// ---- VISUs/AxisControl.TcVIS
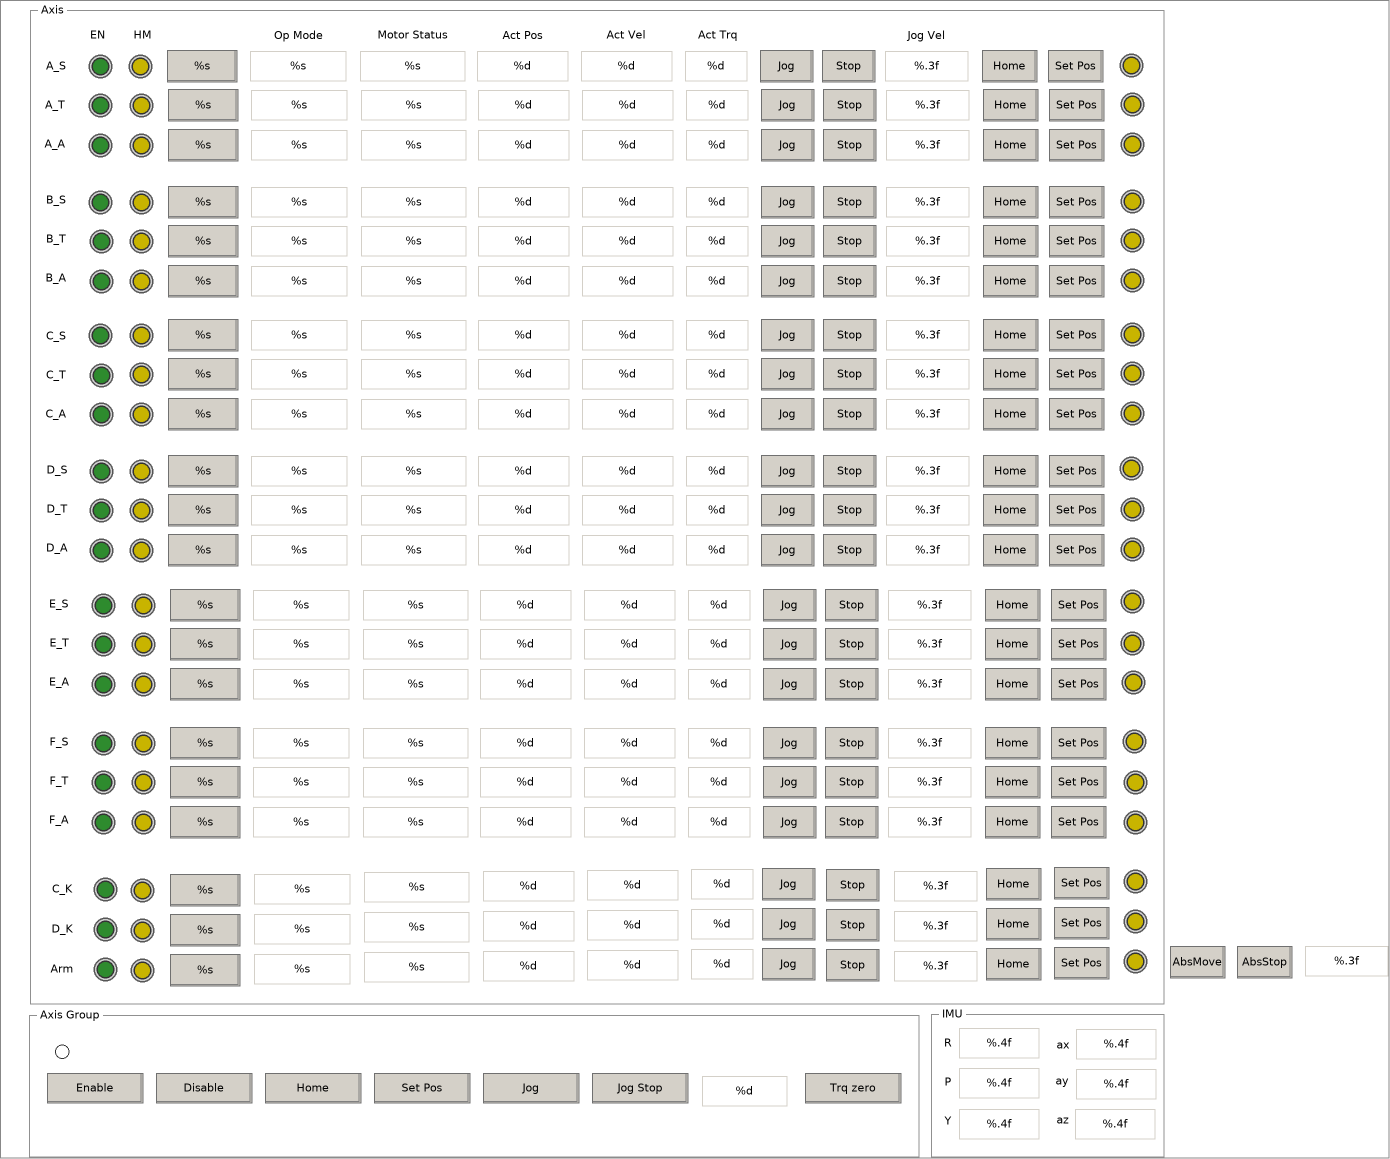
VISUALIZATION AxisControl  // 1390x1159
    GroupBox (30,2 1134x1002), "Axis"
        Label (37,23 61x20), "EN"
        Label (324,25 117x16), "Motor Status"
        Label (239,24 59x19), "Op Mode"
        Label (465,27 55x13), "Act Pos"
        Lamp1 (57,50 27x29), variable: GVL.motorDrive[0].enableBit, style: Lamp-Lamp1-Green
        Textfield (220,49 96x30), "%s", text variable: GVL.motorDrive[0].opModeDispStr
        Textfield (330,49 105x30), "%s", text variable: GVL.motorDrive[0].statusDispStr
        Textfield (447,49 91x30), "%d", text variable: GVL.motorDrive[0].motor.actualPos
        Textfield (551,49 91x30), "%d", text variable: GVL.motorDrive[0].motor.actualVel
        Label (653,25 70x16), "Act Trq"
        Textfield (655,49 62x30), "%d", text variable: GVL.motorDrive[0].motor.actualTrq
        Button (137,48 70x32), "%s", text variable: GVL.enablebuttonText[0]
            toggle GVL.enableButton[0]
        Label (561,25 70x16), "Act Vel"
        Lamp1 (97,50 27x29), variable: GVL.motorDrive[0].isHomeSwitchOn, style: Lamp-Lamp1-Yellow
        Label (91,21 43x24), "HM"
        Button (730,48 53x32), "Jog"
            toggle GVL.jogButton[0]
        Label (869,27 55x13), "Jog Vel"
        Button (952,48 55x32), "Home"
            toggle GVL.startHomeButton[0]
        Button (1018,48 55x32), "Set Pos"
            toggle GVL.setInitPositionButton[0]
        Label (5,54 42x20), "A_S"
        Textfield (855,49 83x30), "%.3f", text variable: GVL.jogVelocity[0]
            OnMouseClick: write the text variable via Default
        Lamp1 (57,89 27x29), variable: GVL.motorDrive[1].enableBit, style: Lamp-Lamp1-Green
        Lamp1 (57,129 27x29), variable: GVL.motorDrive[2].enableBit, style: Lamp-Lamp1-Green
        Lamp1 (57,186 27x29), variable: GVL.motorDrive[3].enableBit, style: Lamp-Lamp1-Green
        Lamp1 (57,319 27x29), variable: GVL.motorDrive[6].enableBit, style: Lamp-Lamp1-Green
        Button (792,48 53x32), "Stop"
            toggle GVL.jogStopButton[0]
        Lamp1 (1088,49 27x29), variable: GVL.motorDrive[0].isHoming, style: Lamp-Lamp1-Yellow
        Lamp1 (1088,452 27x29), variable: GVL.motorDrive[9].isHoming, style: Lamp-Lamp1-Yellow
        Label (8,592 42x20), "E_S"
        Label (8,631 42x20), "E_T"
        Label (8,670 42x20), "E_A"
        Lamp1 (60,589 27x29), variable: GVL.motorDrive[12].enableBit, style: Lamp-Lamp1-Green
        Textfield (223,588 96x30), "%s", text variable: GVL.motorDrive[12].opModeDispStr
        Textfield (333,588 105x30), "%s", text variable: GVL.motorDrive[12].statusDispStr
        Textfield (450,588 91x30), "%d", text variable: GVL.motorDrive[12].motor.actualPos
        Textfield (554,588 91x30), "%d", text variable: GVL.motorDrive[12].motor.actualVel
        Button (140,587 70x32), "%s", text variable: GVL.enablebuttonText[12]
            toggle GVL.enableButton[12]
        Lamp1 (100,589 27x29), variable: GVL.motorDrive[12].isHomeSwitchOn, style: Lamp-Lamp1-Yellow
        Button (733,587 53x32), "Jog"
            toggle GVL.jogButton[12]
        Button (955,587 55x32), "Home"
            toggle GVL.startHomeButton[12]
        Button (1021,587 55x32), "Set Pos"
            toggle GVL.setInitPositionButton[12]
        Textfield (858,588 83x30), "%.3f", text variable: GVL.jogVelocity[12]
            OnMouseClick: write the text variable via Default
        Lamp1 (60,628 27x29), variable: GVL.motorDrive[13].enableBit, style: Lamp-Lamp1-Green
        Lamp1 (60,668 27x29), variable: GVL.motorDrive[14].enableBit, style: Lamp-Lamp1-Green
        Textfield (223,627 96x30), "%s", text variable: GVL.motorDrive[13].opModeDispStr
        Textfield (333,627 105x30), "%s", text variable: GVL.motorDrive[13].statusDispStr
        Textfield (450,627 91x30), "%d", text variable: GVL.motorDrive[13].motor.actualPos
        Textfield (554,627 91x30), "%d", text variable: GVL.motorDrive[13].motor.actualVel
        Textfield (658,627 62x30), "%d", text variable: GVL.motorDrive[13].motor.actualTrq
        Button (140,626 70x32), "%s", text variable: GVL.enablebuttonText[13]
            toggle GVL.enableButton[13]
        Lamp1 (100,628 27x29), variable: GVL.motorDrive[13].isHomeSwitchOn, style: Lamp-Lamp1-Yellow
        Button (733,626 53x32), "Jog"
            toggle GVL.jogButton[13]
        Button (955,626 55x32), "Home"
            toggle GVL.startHomeButton[13]
        Button (1021,626 55x32), "Set Pos"
            toggle GVL.setInitPositionButton[13]
        Textfield (858,627 83x30), "%.3f", text variable: GVL.jogVelocity[13]
            OnMouseClick: write the text variable via Default
        Textfield (223,667 96x30), "%s", text variable: GVL.motorDrive[14].opModeDispStr
        Textfield (333,667 105x30), "%s", text variable: GVL.motorDrive[14].statusDispStr
        Textfield (450,667 91x30), "%d", text variable: GVL.motorDrive[14].motor.actualPos
        Textfield (554,667 91x30), "%d", text variable: GVL.motorDrive[14].motor.actualVel
        Textfield (658,667 62x30), "%d", text variable: GVL.motorDrive[14].motor.actualTrq
        Button (140,666 70x32), "%s", text variable: GVL.enablebuttonText[14]
            toggle GVL.enableButton[14]
        Lamp1 (100,668 27x29), variable: GVL.motorDrive[14].isHomeSwitchOn, style: Lamp-Lamp1-Yellow
        Button (733,666 53x32), "Jog"
            toggle GVL.jogButton[14]
        Button (955,666 55x32), "Home"
            toggle GVL.startHomeButton[14]
        Button (1021,666 55x32), "Set Pos"
            toggle GVL.setInitPositionButton[14]
        Textfield (858,667 83x30), "%.3f", text variable: GVL.jogVelocity[14]
            OnMouseClick: write the text variable via Default
        Button (795,587 53x32), "Stop"
            toggle GVL.jogStopButton[12]
        Button (795,626 53x32), "Stop"
            toggle GVL.jogStopButton[13]
        Button (795,666 53x32), "Stop"
            toggle GVL.jogStopButton[14]
        Label (8,730 42x20), "F_S"
        Label (8,769 42x20), "F_T"
        Label (8,808 42x20), "F_A"
        Lamp1 (60,727 27x29), variable: GVL.motorDrive[15].enableBit, style: Lamp-Lamp1-Green
        Textfield (223,726 96x30), "%s", text variable: GVL.motorDrive[15].opModeDispStr
        Textfield (333,726 105x30), "%s", text variable: GVL.motorDrive[15].statusDispStr
        Textfield (450,726 91x30), "%d", text variable: GVL.motorDrive[15].motor.actualPos
        Textfield (554,726 91x30), "%d", text variable: GVL.motorDrive[15].motor.actualVel
        Textfield (658,726 62x30), "%d", text variable: GVL.motorDrive[15].motor.actualTrq
        Button (140,725 70x32), "%s", text variable: GVL.enablebuttonText[15]
            toggle GVL.enableButton[15]
        Lamp1 (100,727 27x29), variable: GVL.motorDrive[15].isHomeSwitchOn, style: Lamp-Lamp1-Yellow
        Button (733,725 53x32), "Jog"
            toggle GVL.jogButton[15]
        Button (955,725 55x32), "Home"
            toggle GVL.startHomeButton[15]
        Button (1021,725 55x32), "Set Pos"
            toggle GVL.setInitPositionButton[15]
        Textfield (858,726 83x30), "%.3f", text variable: GVL.jogVelocity[15]
            OnMouseClick: write the text variable via Default
        Lamp1 (60,766 27x29), variable: GVL.motorDrive[16].enableBit, style: Lamp-Lamp1-Green
        Lamp1 (60,806 27x29), variable: GVL.motorDrive[17].enableBit, style: Lamp-Lamp1-Green
        Textfield (223,765 96x30), "%s", text variable: GVL.motorDrive[16].opModeDispStr
        Textfield (333,765 105x30), "%s", text variable: GVL.motorDrive[16].statusDispStr
        Textfield (450,765 91x30), "%d", text variable: GVL.motorDrive[16].motor.actualPos
        Textfield (554,765 91x30), "%d", text variable: GVL.motorDrive[16].motor.actualVel
        Textfield (658,765 62x30), "%d", text variable: GVL.motorDrive[16].motor.actualTrq
        Button (140,764 70x32), "%s", text variable: GVL.enablebuttonText[16]
            toggle GVL.enableButton[16]
        Lamp1 (100,766 27x29), variable: GVL.motorDrive[16].isHomeSwitchOn, style: Lamp-Lamp1-Yellow
        Button (733,764 53x32), "Jog"
            toggle GVL.jogButton[16]
        Button (955,764 55x32), "Home"
            toggle GVL.startHomeButton[16]
        Button (1021,764 55x32), "Set Pos"
            toggle GVL.setInitPositionButton[16]
        Textfield (858,765 83x30), "%.3f", text variable: GVL.jogVelocity[16]
            OnMouseClick: write the text variable via Default
        Textfield (223,805 96x30), "%s", text variable: GVL.motorDrive[17].opModeDispStr
        Textfield (333,805 105x30), "%s", text variable: GVL.motorDrive[17].statusDispStr
        Textfield (450,805 91x30), "%d", text variable: GVL.motorDrive[17].motor.actualPos
        Textfield (554,805 91x30), "%d", text variable: GVL.motorDrive[17].motor.actualVel
        Textfield (658,805 62x30), "%d", text variable: GVL.motorDrive[17].motor.actualTrq
        Button (140,804 70x32), "%s", text variable: GVL.enablebuttonText[17]
            toggle GVL.enableButton[17]
        Lamp1 (100,806 27x29), variable: GVL.motorDrive[17].isHomeSwitchOn, style: Lamp-Lamp1-Yellow
        Button (733,804 53x32), "Jog"
            toggle GVL.jogButton[17]
        Button (955,804 55x32), "Home"
            toggle GVL.startHomeButton[17]
        Button (1021,804 55x32), "Set Pos"
            toggle GVL.setInitPositionButton[17]
        Textfield (858,805 83x30), "%.3f", text variable: GVL.jogVelocity[17]
            OnMouseClick: write the text variable via Default
        Button (795,725 53x32), "Stop"
            toggle GVL.jogStopButton[15]
        Button (795,764 53x32), "Stop"
            toggle GVL.jogStopButton[16]
        Button (795,804 53x32), "Stop"
            toggle GVL.jogStopButton[17]
        Lamp1 (1089,585 27x29), variable: GVL.motorDrive[12].isHoming, style: Lamp-Lamp1-Yellow
        Lamp1 (1091,725 27x29), variable: GVL.motorDrive[15].isHoming, style: Lamp-Lamp1-Yellow
        Lamp1 (1092,766 27x29), variable: GVL.motorDrive[16].isHoming, style: Lamp-Lamp1-Yellow
        Lamp1 (1092,806 27x29), variable: GVL.motorDrive[17].isHoming, style: Lamp-Lamp1-Yellow
        Lamp1 (1089,627 27x29), variable: GVL.motorDrive[13].isHoming, style: Lamp-Lamp1-Yellow
        Label (11,877 42x20), "C_K"
        Lamp1 (62,873 27x29), variable: GVL.motorDrive[18].enableBit, style: Lamp-Lamp1-Green
        Lamp1 (99,874 27x29), variable: GVL.motorDrive[18].isHomeSwitchOn, style: Lamp-Lamp1-Yellow
        Button (140,872 70x32), "%s", text variable: GVL.enablebuttonText[17]
            toggle GVL.enableButton[18]
        Textfield (224,872 96x30), "%s", text variable: GVL.motorDrive[18].opModeDispStr
        Textfield (334,870 105x30), "%s", text variable: GVL.motorDrive[18].statusDispStr
        Textfield (453,869 91x30), "%d", text variable: GVL.motorDrive[18].motor.actualPos
        Textfield (557,868 91x30), "%d", text variable: GVL.motorDrive[18].motor.actualVel
        Textfield (661,867 62x30), "%d", text variable: GVL.motorDrive[18].motor.actualTrq
        Button (732,866 53x32), "Jog"
            toggle GVL.jogButton[18]
        Button (796,867 53x32), "Stop"
            toggle GVL.jogStopButton[18]
        Textfield (864,869 83x30), "%.3f", text variable: GVL.jogVelocity[18]
            OnMouseClick: write the text variable via Default
        Button (956,866 55x32), "Home"
            toggle GVL.startHomeButton[18]
        Button (1024,865 55x32), "Set Pos"
            toggle GVL.setInitPositionButton[18]
        Lamp1 (1092,865 27x29), variable: GVL.motorDrive[18].isHoming, style: Lamp-Lamp1-Yellow
        Textfield (658,588 62x30), "%d", text variable: GVL.motorDrive[12].motor.actualTrq
        Label (11,917 42x20), "D_K"
        Label (11,957 42x20), "Arm"
    Label (34,95 42x20), "A_T"
    Label (34,134 42x20), "A_A"
    Label (35,190 42x20), "B_S"
    Label (35,229 42x20), "B_T"
    Label (35,268 42x20), "B_A"
    Label (35,326 42x20), "C_S"
    Label (35,365 42x20), "C_T"
    Label (35,404 42x20), "C_A"
    Label (36,460 42x20), "D_S"
    Label (36,499 42x20), "D_T"
    Label (36,538 42x20), "D_A"
    GroupBox (29,1007 890x150), "Axis Group"
        RadioButton (24,30 783x29), variable: GVL.groupSelector
            Areas[1]: Text=Shank
            Areas[2]: Text=Thigh
            Areas[3]: Text=Side
            Areas[4]: Text=LegA
            Areas[5]: Text=LegB
            Areas[6]: Text=LegC
            Areas[7]: Text=LegD
            Areas[8]: Text=LegE
            Areas[9]: Text=LegF
        Button (18,66 96x30), "Enable"
            toggle GVL.enableGroupButton
        Button (127,66 96x30), "Disable"
            toggle GVL.disableGroupButton
        Button (236,66 96x30), "Home"
            toggle GVL.homeGroupButton
        Button (345,66 96x30), "Set Pos"
            toggle GVL.setPosGroupButton
        Button (454,66 96x30), "Jog"
            toggle GVL.jogGroupButton
        Button (776,66 96x30), "Trq zero"
            toggle GVL.setTSRZeroButton
        Textfield (673,69 85x30), "%d", text variable: GVL.jogGroupVelocity
            OnMouseClick: write the text variable via Default
        Button (563,66 96x30), "Jog Stop"
            toggle GVL.jogStopGroupButton
    Textfield (251,90 96x30), "%s", text variable: GVL.motorDrive[1].opModeDispStr
    Textfield (361,90 105x30), "%s", text variable: GVL.motorDrive[1].statusDispStr
    Textfield (478,90 91x30), "%d", text variable: GVL.motorDrive[1].motor.actualPos
    Textfield (582,90 91x30), "%d", text variable: GVL.motorDrive[1].motor.actualVel
    Textfield (686,90 62x30), "%d", text variable: GVL.motorDrive[1].motor.actualTrq
    Button (168,89 70x32), "%s", text variable: GVL.enablebuttonText[1]
        toggle GVL.enableButton[1]
    Lamp1 (128,91 27x29), variable: GVL.motorDrive[1].isHomeSwitchOn, style: Lamp-Lamp1-Yellow
    Button (761,89 53x32), "Jog"
        toggle GVL.jogButton[1]
    Button (983,89 55x32), "Home"
        toggle GVL.startHomeButton[1]
    Button (1049,89 55x32), "Set Pos"
        toggle GVL.setInitPositionButton[1]
    Textfield (886,90 83x30), "%.3f", text variable: GVL.jogVelocity[1]
        OnMouseClick: write the text variable via Default
    Textfield (251,130 96x30), "%s", text variable: GVL.motorDrive[2].opModeDispStr
    Textfield (361,130 105x30), "%s", text variable: GVL.motorDrive[2].statusDispStr
    Textfield (478,130 91x30), "%d", text variable: GVL.motorDrive[2].motor.actualPos
    Textfield (582,130 91x30), "%d", text variable: GVL.motorDrive[2].motor.actualVel
    Textfield (686,130 62x30), "%d", text variable: GVL.motorDrive[2].motor.actualTrq
    Button (168,129 70x32), "%s", text variable: GVL.enablebuttonText[2]
        toggle GVL.enableButton[2]
    Lamp1 (128,131 27x29), variable: GVL.motorDrive[2].isHomeSwitchOn, style: Lamp-Lamp1-Yellow
    Button (761,129 53x32), "Jog"
        toggle GVL.jogButton[2]
    Button (983,129 55x32), "Home"
        toggle GVL.startHomeButton[2]
    Button (1049,129 55x32), "Set Pos"
        toggle GVL.setInitPositionButton[2]
    Textfield (886,130 83x30), "%.3f", text variable: GVL.jogVelocity[2]
        OnMouseClick: write the text variable via Default
    Textfield (251,187 96x30), "%s", text variable: GVL.motorDrive[3].opModeDispStr
    Textfield (361,187 105x30), "%s", text variable: GVL.motorDrive[3].statusDispStr
    Textfield (478,187 91x30), "%d", text variable: GVL.motorDrive[3].motor.actualPos
    Textfield (582,187 91x30), "%d", text variable: GVL.motorDrive[3].motor.actualVel
    Textfield (686,187 62x30), "%d", text variable: GVL.motorDrive[3].motor.actualTrq
    Button (168,186 70x32), "%s", text variable: GVL.enablebuttonText[3]
        toggle GVL.enableButton[3]
    Lamp1 (128,188 27x29), variable: GVL.motorDrive[3].isHomeSwitchOn, style: Lamp-Lamp1-Yellow
    Button (761,186 53x32), "Jog"
        toggle GVL.jogButton[3]
    Button (983,186 55x32), "Home"
        toggle GVL.startHomeButton[3]
    Button (1049,186 55x32), "Set Pos"
        toggle GVL.setInitPositionButton[3]
    Textfield (886,187 83x30), "%.3f", text variable: GVL.jogVelocity[3]
        OnMouseClick: write the text variable via Default
    Lamp1 (88,227 27x29), variable: GVL.motorDrive[4].enableBit, style: Lamp-Lamp1-Green
    Lamp1 (88,267 27x29), variable: GVL.motorDrive[5].enableBit, style: Lamp-Lamp1-Green
    Textfield (251,226 96x30), "%s", text variable: GVL.motorDrive[4].opModeDispStr
    Textfield (361,226 105x30), "%s", text variable: GVL.motorDrive[4].statusDispStr
    Textfield (478,226 91x30), "%d", text variable: GVL.motorDrive[4].motor.actualPos
    Textfield (582,226 91x30), "%d", text variable: GVL.motorDrive[4].motor.actualVel
    Textfield (686,226 62x30), "%d", text variable: GVL.motorDrive[4].motor.actualTrq
    Button (168,225 70x32), "%s", text variable: GVL.enablebuttonText[4]
        toggle GVL.enableButton[4]
    Lamp1 (128,227 27x29), variable: GVL.motorDrive[4].isHomeSwitchOn, style: Lamp-Lamp1-Yellow
    Button (761,225 53x32), "Jog"
        toggle GVL.jogButton[4]
    Button (983,225 55x32), "Home"
        toggle GVL.startHomeButton[4]
    Button (1049,225 55x32), "Set Pos"
        toggle GVL.setInitPositionButton[4]
    Textfield (886,226 83x30), "%.3f", text variable: GVL.jogVelocity[4]
        OnMouseClick: write the text variable via Default
    Textfield (251,266 96x30), "%s", text variable: GVL.motorDrive[5].opModeDispStr
    Textfield (361,266 105x30), "%s", text variable: GVL.motorDrive[5].statusDispStr
    Textfield (478,266 91x30), "%d", text variable: GVL.motorDrive[5].motor.actualPos
    Textfield (582,266 91x30), "%d", text variable: GVL.motorDrive[5].motor.actualVel
    Textfield (686,266 62x30), "%d", text variable: GVL.motorDrive[5].motor.actualTrq
    Button (168,265 70x32), "%s", text variable: GVL.enablebuttonText[5]
        toggle GVL.enableButton[5]
    Lamp1 (128,267 27x29), variable: GVL.motorDrive[5].isHomeSwitchOn, style: Lamp-Lamp1-Yellow
    Button (761,265 53x32), "Jog"
        toggle GVL.jogButton[5]
    Button (983,265 55x32), "Home"
        toggle GVL.startHomeButton[5]
    Button (1049,265 55x32), "Set Pos"
        toggle GVL.setInitPositionButton[5]
    Textfield (886,266 83x30), "%.3f", text variable: GVL.jogVelocity[5]
        OnMouseClick: write the text variable via Default
    Textfield (251,320 96x30), "%s", text variable: GVL.motorDrive[6].opModeDispStr
    Textfield (361,320 105x30), "%s", text variable: GVL.motorDrive[6].statusDispStr
    Textfield (478,320 91x30), "%d", text variable: GVL.motorDrive[6].motor.actualPos
    Textfield (582,320 91x30), "%d", text variable: GVL.motorDrive[6].motor.actualVel
    Textfield (686,320 62x30), "%d", text variable: GVL.motorDrive[6].motor.actualTrq
    Button (168,319 70x32), "%s", text variable: GVL.enablebuttonText[6]
        toggle GVL.enableButton[6]
    Lamp1 (128,321 27x29), variable: GVL.motorDrive[6].isHomeSwitchOn, style: Lamp-Lamp1-Yellow
    Button (761,319 53x32), "Jog"
        toggle GVL.jogButton[6]
    Button (983,319 55x32), "Home"
        toggle GVL.startHomeButton[6]
    Button (1049,319 55x32), "Set Pos"
        toggle GVL.setInitPositionButton[6]
    Textfield (886,320 83x30), "%.3f", text variable: GVL.jogVelocity[6]
        OnMouseClick: write the text variable via Default
    Lamp1 (88,361 27x29), variable: GVL.motorDrive[7].enableBit, style: Lamp-Lamp1-Green
    Lamp1 (88,400 27x29), variable: GVL.motorDrive[8].enableBit, style: Lamp-Lamp1-Green
    Lamp1 (88,457 27x29), variable: GVL.motorDrive[9].enableBit, style: Lamp-Lamp1-Green
    Textfield (251,359 96x30), "%s", text variable: GVL.motorDrive[7].opModeDispStr
    Textfield (361,359 105x30), "%s", text variable: GVL.motorDrive[7].statusDispStr
    Textfield (478,359 91x30), "%d", text variable: GVL.motorDrive[7].motor.actualPos
    Textfield (582,359 91x30), "%d", text variable: GVL.motorDrive[7].motor.actualVel
    Textfield (686,359 62x30), "%d", text variable: GVL.motorDrive[7].motor.actualTrq
    Button (168,358 70x32), "%s", text variable: GVL.enablebuttonText[7]
        toggle GVL.enableButton[7]
    Lamp1 (128,360 27x29), variable: GVL.motorDrive[7].isHomeSwitchOn, style: Lamp-Lamp1-Yellow
    Button (761,358 53x32), "Jog"
        toggle GVL.jogButton[7]
    Button (983,358 55x32), "Home"
        toggle GVL.startHomeButton[7]
    Button (1049,358 55x32), "Set Pos"
        toggle GVL.setInitPositionButton[7]
    Textfield (886,359 83x30), "%.3f", text variable: GVL.jogVelocity[7]
        OnMouseClick: write the text variable via Default
    Textfield (251,399 96x30), "%s", text variable: GVL.motorDrive[8].opModeDispStr
    Textfield (361,399 105x30), "%s", text variable: GVL.motorDrive[8].statusDispStr
    Textfield (478,399 91x30), "%d", text variable: GVL.motorDrive[8].motor.actualPos
    Textfield (582,399 91x30), "%d", text variable: GVL.motorDrive[8].motor.actualVel
    Textfield (686,399 62x30), "%d", text variable: GVL.motorDrive[8].motor.actualTrq
    Button (168,398 70x32), "%s", text variable: GVL.enablebuttonText[8]
        toggle GVL.enableButton[8]
    Lamp1 (128,400 27x29), variable: GVL.motorDrive[8].isHomeSwitchOn, style: Lamp-Lamp1-Yellow
    Button (761,398 53x32), "Jog"
        toggle GVL.jogButton[8]
    Button (983,398 55x32), "Home"
        toggle GVL.startHomeButton[8]
    Button (1049,398 55x32), "Set Pos"
        toggle GVL.setInitPositionButton[8]
    Textfield (886,399 83x30), "%.3f", text variable: GVL.jogVelocity[8]
        OnMouseClick: write the text variable via Default
    Textfield (251,456 96x30), "%s", text variable: GVL.motorDrive[9].opModeDispStr
    Textfield (361,456 105x30), "%s", text variable: GVL.motorDrive[9].statusDispStr
    Textfield (478,456 91x30), "%d", text variable: GVL.motorDrive[9].motor.actualPos
    Textfield (582,456 91x30), "%d", text variable: GVL.motorDrive[9].motor.actualVel
    Textfield (686,456 62x30), "%d", text variable: GVL.motorDrive[9].motor.actualTrq
    Button (168,455 70x32), "%s", text variable: GVL.enablebuttonText[9]
        toggle GVL.enableButton[9]
    Lamp1 (128,457 27x29), variable: GVL.motorDrive[9].isHomeSwitchOn, style: Lamp-Lamp1-Yellow
    Button (761,455 53x32), "Jog"
        toggle GVL.jogButton[9]
    Button (983,455 55x32), "Home"
        toggle GVL.startHomeButton[9]
    Button (1049,455 55x32), "Set Pos"
        toggle GVL.setInitPositionButton[9]
    Textfield (886,456 83x30), "%.3f", text variable: GVL.jogVelocity[9]
        OnMouseClick: write the text variable via Default
    Lamp1 (88,496 27x29), variable: GVL.motorDrive[10].enableBit, style: Lamp-Lamp1-Green
    Lamp1 (88,536 27x29), variable: GVL.motorDrive[11].enableBit, style: Lamp-Lamp1-Green
    Textfield (251,495 96x30), "%s", text variable: GVL.motorDrive[10].opModeDispStr
    Textfield (361,495 105x30), "%s", text variable: GVL.motorDrive[10].statusDispStr
    Textfield (478,495 91x30), "%d", text variable: GVL.motorDrive[10].motor.actualPos
    Textfield (582,495 91x30), "%d", text variable: GVL.motorDrive[10].motor.actualVel
    Textfield (686,495 62x30), "%d", text variable: GVL.motorDrive[10].motor.actualTrq
    Button (168,494 70x32), "%s", text variable: GVL.enablebuttonText[10]
        toggle GVL.enableButton[10]
    Lamp1 (128,496 27x29), variable: GVL.motorDrive[10].isHomeSwitchOn, style: Lamp-Lamp1-Yellow
    Button (761,494 53x32), "Jog"
        toggle GVL.jogButton[10]
    Button (983,494 55x32), "Home"
        toggle GVL.startHomeButton[10]
    Button (1049,494 55x32), "Set Pos"
        toggle GVL.setInitPositionButton[10]
    Textfield (886,495 83x30), "%.3f", text variable: GVL.jogVelocity[10]
        OnMouseClick: write the text variable via Default
    Textfield (251,535 96x30), "%s", text variable: GVL.motorDrive[11].opModeDispStr
    Textfield (361,535 105x30), "%s", text variable: GVL.motorDrive[11].statusDispStr
    Textfield (478,535 91x30), "%d", text variable: GVL.motorDrive[11].motor.actualPos
    Textfield (582,535 91x30), "%d", text variable: GVL.motorDrive[11].motor.actualVel
    Textfield (686,535 62x30), "%d", text variable: GVL.motorDrive[11].motor.actualTrq
    Button (168,534 70x32), "%s", text variable: GVL.enablebuttonText[11]
        toggle GVL.enableButton[11]
    Lamp1 (128,536 27x29), variable: GVL.motorDrive[11].isHomeSwitchOn, style: Lamp-Lamp1-Yellow
    Button (761,534 53x32), "Jog"
        toggle GVL.jogButton[11]
    Button (983,534 55x32), "Home"
        toggle GVL.startHomeButton[11]
    Button (1049,534 55x32), "Set Pos"
        toggle GVL.setInitPositionButton[11]
    Textfield (886,535 83x30), "%.3f", text variable: GVL.jogVelocity[11]
        OnMouseClick: write the text variable via Default
    Button (823,89 53x32), "Stop"
        toggle GVL.jogStopButton[1]
    Button (823,129 53x32), "Stop"
        toggle GVL.jogStopButton[2]
    Button (823,186 53x32), "Stop"
        toggle GVL.jogStopButton[3]
    Button (823,225 53x32), "Stop"
        toggle GVL.jogStopButton[4]
    Button (823,265 53x32), "Stop"
        toggle GVL.jogStopButton[5]
    Button (823,319 53x32), "Stop"
        toggle GVL.jogStopButton[6]
    Button (823,358 53x32), "Stop"
        toggle GVL.jogStopButton[7]
    Button (823,398 53x32), "Stop"
        toggle GVL.jogStopButton[8]
    Button (823,455 53x32), "Stop"
        toggle GVL.jogStopButton[9]
    Button (823,494 53x32), "Stop"
        toggle GVL.jogStopButton[10]
    Button (823,534 53x32), "Stop"
        toggle GVL.jogStopButton[11]
    Lamp1 (1119,90 27x29), variable: GVL.motorDrive[1].isHoming, style: Lamp-Lamp1-Yellow
    Lamp1 (1119,130 27x29), variable: GVL.motorDrive[2].isHoming, style: Lamp-Lamp1-Yellow
    Lamp1 (1119,187 27x29), variable: GVL.motorDrive[3].isHoming, style: Lamp-Lamp1-Yellow
    Lamp1 (1119,226 27x29), variable: GVL.motorDrive[4].isHoming, style: Lamp-Lamp1-Yellow
    Lamp1 (1119,266 27x29), variable: GVL.motorDrive[5].isHoming, style: Lamp-Lamp1-Yellow
    Lamp1 (1119,320 27x29), variable: GVL.motorDrive[6].isHoming, style: Lamp-Lamp1-Yellow
    Lamp1 (1119,359 27x29), variable: GVL.motorDrive[7].isHoming, style: Lamp-Lamp1-Yellow
    Lamp1 (1119,399 27x29), variable: GVL.motorDrive[8].isHoming, style: Lamp-Lamp1-Yellow
    Lamp1 (1119,495 27x29), variable: GVL.motorDrive[10].isHoming, style: Lamp-Lamp1-Yellow
    Lamp1 (1119,535 27x29), variable: GVL.motorDrive[11].isHoming, style: Lamp-Lamp1-Yellow
    Lamp1 (1120,668 27x29), variable: GVL.motorDrive[14].isHoming, style: Lamp-Lamp1-Yellow
    GroupBox (931,1006 233x151), "IMU"
        Textfield (28,22 80x30), "%.4f", text variable: GVL.rpy_model[0]
        Textfield (28,62 80x30), "%.4f", text variable: GVL.rpy_model[1]
        Textfield (28,103 80x30), "%.4f", text variable: GVL.rpy_model[2]
        Label (-5,22 44x30), "R"
        Label (-5,61 44x30), "P"
        Label (-5,100 44x30), "Y"
        Textfield (145,23 80x30), "%.4f", text variable: GVL.accx
        Label (110,24 44x30), "ax"
        Textfield (145,63 80x30), "%.4f", text variable: GVL.accy
        Label (109,60 44x30), "ay"
        Label (110,99 44x30), "az"
        Textfield (144,103 80x30), "%.4f", text variable: GVL.accz
    Lamp1 (92,915 27x29), variable: GVL.motorDrive[19].enableBit, style: Lamp-Lamp1-Green
    Lamp1 (129,916 27x29), variable: GVL.motorDrive[19].isHomeSwitchOn, style: Lamp-Lamp1-Yellow
    Button (170,914 70x32), "%s", text variable: GVL.enablebuttonText[17]
        toggle GVL.enableButton[19]
    Textfield (254,914 96x30), "%s", text variable: GVL.motorDrive[19].opModeDispStr
    Textfield (364,912 105x30), "%s", text variable: GVL.motorDrive[19].statusDispStr
    Textfield (483,911 91x30), "%d", text variable: GVL.motorDrive[19].motor.actualPos
    Textfield (587,910 91x30), "%d", text variable: GVL.motorDrive[19].motor.actualVel
    Textfield (691,909 62x30), "%d", text variable: GVL.motorDrive[19].motor.actualTrq
    Button (762,908 53x32), "Jog"
        toggle GVL.jogButton[19]
    Button (826,909 53x32), "Stop"
        toggle GVL.jogStopButton[19]
    Textfield (894,911 83x30), "%.3f", text variable: GVL.jogVelocity[19]
        OnMouseClick: write the text variable via Default
    Button (986,908 55x32), "Home"
        toggle GVL.startHomeButton[19]
    Button (1054,907 55x32), "Set Pos"
        toggle GVL.setInitPositionButton[19]
    Lamp1 (1122,907 27x29), variable: GVL.motorDrive[19].isHoming, style: Lamp-Lamp1-Yellow
    Lamp1 (92,955 27x29), variable: GVL.motorDrive[20].enableBit, style: Lamp-Lamp1-Green
    Lamp1 (129,956 27x29), variable: GVL.motorDrive[20].isHomeSwitchOn, style: Lamp-Lamp1-Yellow
    Button (170,954 70x32), "%s", text variable: GVL.enablebuttonText[17]
        toggle GVL.enableButton[20]
    Textfield (254,954 96x30), "%s", text variable: GVL.motorDrive[20].opModeDispStr
    Textfield (364,952 105x30), "%s", text variable: GVL.motorDrive[20].statusDispStr
    Textfield (483,951 91x30), "%d", text variable: GVL.motorDrive[20].motor.actualPos
    Textfield (587,950 91x30), "%d", text variable: GVL.motorDrive[20].motor.actualVel
    Textfield (691,949 62x30), "%d", text variable: GVL.motorDrive[20].motor.actualTrq
    Button (762,948 53x32), "Jog"
        toggle GVL.jogButton[20]
    Button (826,949 53x32), "Stop"
        toggle GVL.jogStopButton[20]
    Textfield (894,951 83x30), "%.3f", text variable: GVL.jogVelocity[20]
        OnMouseClick: write the text variable via Default
    Button (986,948 55x32), "Home"
        toggle GVL.startHomeButton[20]
    Button (1054,947 55x32), "Set Pos"
        toggle GVL.setInitPositionButton[20]
    Lamp1 (1122,947 27x29), variable: GVL.motorDrive[20].isHoming, style: Lamp-Lamp1-Yellow
    Button (1170,946 55x32), "AbsMove"
        toggle GVL.AbsMoveButton[20]
    Textfield (1305,946 83x30), "%.3f", text variable: GVL.AbsMoveTgtPos[20]
        OnMouseClick: write the text variable via Default
    Button (1237,946 55x32), "AbsStop"
        toggle GVL.AbsMoveStopButton[20]
END_VISUALIZATION

// ---- VISUs/ForceControl.TcVIS
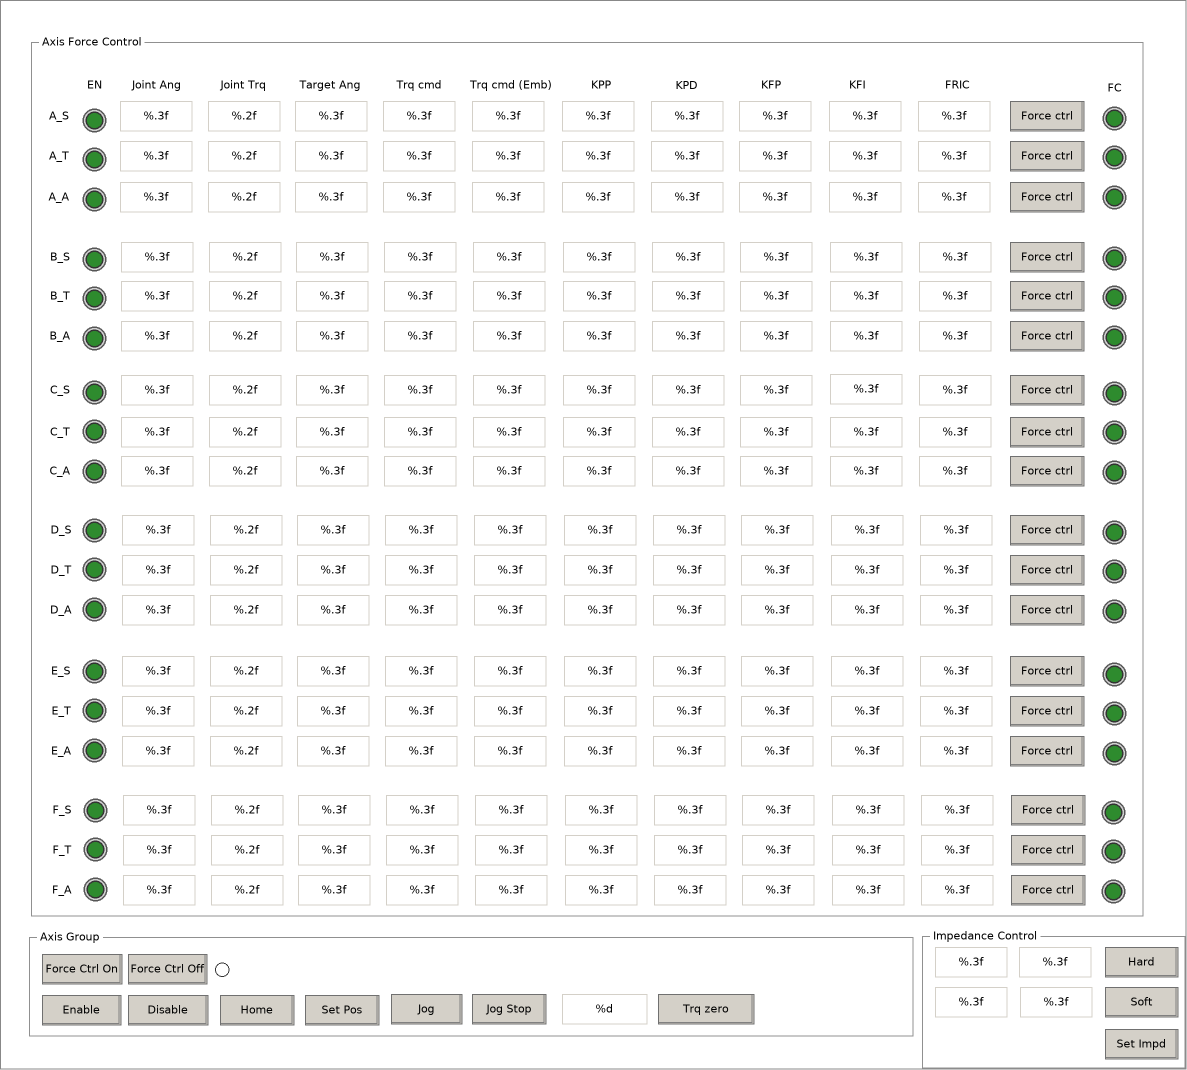
VISUALIZATION ForceControl  // 1187x1070
    GroupBox (31,34 1112x882), "Axis Force Control"
        Label (90,36 71x30), "Joint Ang"
        Label (179,36 67x30), "Joint Trq"
        Label (263,36 72x30), "Target Ang"
        Label (353,36 70x30), "Trq cmd"
        Label (433,36 94x30), "Trq cmd (Emb)"
        Textfield (89,67 72x30), "%.3f", text variable: GVL.motorDrive[0].motorAngle
        Label (545,39 50x24), "KPP"
        Label (632,36 47x31), "KPD"
        Label (800,36 53x30), "KFI"
        Label (714,36 52x30), "KFP"
        Label (900,36 53x30), "FRIC"
        Label (7,72 42x20), "A_S"
        Label (7,112 42x20), "A_T"
        Label (7,153 42x20), "A_A"
        Label (8,213 42x20), "B_S"
        Label (8,252 42x20), "B_T"
        Label (8,292 42x20), "B_A"
        Label (8,346 42x20), "C_S"
        Label (8,388 42x20), "C_T"
        Label (8,427 42x20), "C_A"
        Label (9,486 42x20), "D_S"
        Label (9,526 42x20), "D_T"
        Label (9,566 42x20), "D_A"
        Textfield (89,107 72x30), "%.3f", text variable: GVL.motorDrive[1].motorAngle
        Textfield (89,148 72x30), "%.3f", text variable: GVL.motorDrive[2].motorAngle
        Textfield (90,208 72x30), "%.3f", text variable: GVL.motorDrive[3].motorAngle
        Textfield (90,247 72x30), "%.3f", text variable: GVL.motorDrive[4].motorAngle
        Textfield (90,287 72x30), "%.3f", text variable: GVL.motorDrive[5].motorAngle
        Textfield (91,481 72x30), "%.3f", text variable: GVL.motorDrive[9].motorAngle
        Textfield (177,67 72x30), "%.2f", text variable: GVL.motorDrive[0].trqCalibrated
        Textfield (264,67 72x30), "%.3f", text variable: GVL.motorDrive[0].tgtAngle
            OnMouseClick: write the text variable via Default
        Textfield (352,67 72x30), "%.3f", text variable: GVL.motorDrive[0].trqOutput
        Button (979,67 74x30), "Force ctrl"
            toggle GVL.axisForceCtrlButton[0]
        Button (979,107 74x30), "Force ctrl"
            toggle GVL.axisForceCtrlButton[1]
        Button (979,148 74x30), "Force ctrl"
            toggle GVL.axisForceCtrlButton[2]
        Button (979,208 74x30), "Force ctrl"
            toggle GVL.axisForceCtrlButton[3]
        Button (979,247 74x30), "Force ctrl"
            toggle GVL.axisForceCtrlButton[4]
        Button (979,287 74x30), "Force ctrl"
            toggle GVL.axisForceCtrlButton[5]
        Button (979,341 74x30), "Force ctrl"
            toggle GVL.axisForceCtrlButton[6]
        Button (979,383 74x30), "Force ctrl"
            toggle GVL.axisForceCtrlButton[7]
        Button (979,422 74x30), "Force ctrl"
            toggle GVL.axisForceCtrlButton[8]
        Button (979,481 74x30), "Force ctrl"
            toggle GVL.axisForceCtrlButton[9]
        Button (979,521 74x30), "Force ctrl"
            toggle GVL.axisForceCtrlButton[10]
        Button (979,561 74x30), "Force ctrl"
            toggle GVL.axisForceCtrlButton[11]
        Textfield (620,67 72x30), "%.3f", text variable: GVL.motorDrive[0].bVirtual
            OnMouseClick: write the text variable via Default
        Textfield (708,67 72x30), "%.3f", text variable: GVL.motorDrive[0].kpTrqLoop
            OnMouseClick: write the text variable via Default
        Textfield (798,67 72x30), "%.3f", text variable: GVL.motorDrive[0].kiTrqLoop
            OnMouseClick: write the text variable via Default
        Textfield (887,67 72x30), "%.3f", text variable: GVL.motorDrive[0].reducerColbConstant
            OnMouseClick: write the text variable via Default
        Lamp1 (1070,70 27x29), variable: GVL.axisForceCtrlModeInd[0], style: Lamp-Lamp1-Green
        Label (1057,39 53x30), "FC"
        Label (33,41 61x20), "EN"
        Label (9,627 42x20), "E_S"
        Label (10,766 42x20), "F_S"
        Lamp1 (1070,626 27x29), variable: GVL.axisForceCtrlModeInd[12], style: Lamp-Lamp1-Green
        Lamp1 (1069,764 27x29), variable: GVL.axisForceCtrlModeInd[15], style: Lamp-Lamp1-Green
        Lamp1 (1069,803 27x29), variable: GVL.axisForceCtrlModeInd[16], style: Lamp-Lamp1-Green
        Lamp1 (1069,843 27x29), variable: GVL.axisForceCtrlModeInd[17], style: Lamp-Lamp1-Green
    Textfield (121,375 72x30), "%.3f", text variable: GVL.motorDrive[6].motorAngle
    Textfield (121,417 72x30), "%.3f", text variable: GVL.motorDrive[7].motorAngle
    Textfield (121,456 72x30), "%.3f", text variable: GVL.motorDrive[8].motorAngle
    Textfield (122,555 72x30), "%.3f", text variable: GVL.motorDrive[10].motorAngle
    Textfield (122,595 72x30), "%.3f", text variable: GVL.motorDrive[11].motorAngle
    Textfield (208,141 72x30), "%.2f", text variable: GVL.motorDrive[1].trqCalibrated
    Textfield (208,182 72x30), "%.2f", text variable: GVL.motorDrive[2].trqCalibrated
    Textfield (209,242 72x30), "%.2f", text variable: GVL.motorDrive[3].trqCalibrated
    Textfield (209,281 72x30), "%.2f", text variable: GVL.motorDrive[4].trqCalibrated
    Textfield (209,321 72x30), "%.2f", text variable: GVL.motorDrive[5].trqCalibrated
    Textfield (210,515 72x30), "%.2f", text variable: GVL.motorDrive[9].trqCalibrated
    Textfield (209,375 72x30), "%.2f", text variable: GVL.motorDrive[6].trqCalibrated
    Textfield (209,417 72x30), "%.2f", text variable: GVL.motorDrive[7].trqCalibrated
    Textfield (209,456 72x30), "%.2f", text variable: GVL.motorDrive[8].trqCalibrated
    Textfield (210,555 72x30), "%.2f", text variable: GVL.motorDrive[10].trqCalibrated
    Textfield (210,595 72x30), "%.2f", text variable: GVL.motorDrive[11].trqCalibrated
    Textfield (295,141 72x30), "%.3f", text variable: GVL.motorDrive[1].tgtAngle
        OnMouseClick: write the text variable via Default
    Textfield (295,182 72x30), "%.3f", text variable: GVL.motorDrive[2].tgtAngle
        OnMouseClick: write the text variable via Default
    Textfield (296,242 72x30), "%.3f", text variable: GVL.motorDrive[3].tgtAngle
        OnMouseClick: write the text variable via Default
    Textfield (296,281 72x30), "%.3f", text variable: GVL.motorDrive[4].tgtAngle
        OnMouseClick: write the text variable via Default
    Textfield (296,321 72x30), "%.3f", text variable: GVL.motorDrive[5].tgtAngle
        OnMouseClick: write the text variable via Default
    Textfield (297,515 72x30), "%.3f", text variable: GVL.motorDrive[9].tgtAngle
        OnMouseClick: write the text variable via Default
    Textfield (296,375 72x30), "%.3f", text variable: GVL.motorDrive[6].tgtAngle
        OnMouseClick: write the text variable via Default
    Textfield (296,417 72x30), "%.3f", text variable: GVL.motorDrive[7].tgtAngle
        OnMouseClick: write the text variable via Default
    Textfield (296,456 72x30), "%.3f", text variable: GVL.motorDrive[8].tgtAngle
        OnMouseClick: write the text variable via Default
    Textfield (297,555 72x30), "%.3f", text variable: GVL.motorDrive[10].tgtAngle
        OnMouseClick: write the text variable via Default
    Textfield (297,595 72x30), "%.3f", text variable: GVL.motorDrive[11].tgtAngle
        OnMouseClick: write the text variable via Default
    Textfield (383,141 72x30), "%.3f", text variable: GVL.motorDrive[1].trqOutput
    Textfield (383,182 72x30), "%.3f", text variable: GVL.motorDrive[2].trqOutput
    Textfield (384,242 72x30), "%.3f", text variable: GVL.motorDrive[3].trqOutput
    Textfield (384,281 72x30), "%.3f", text variable: GVL.motorDrive[4].trqOutput
    Textfield (384,321 72x30), "%.3f", text variable: GVL.motorDrive[5].trqOutput
    Textfield (385,515 72x30), "%.3f", text variable: GVL.motorDrive[9].trqOutput
    Textfield (472,101 72x30), "%.3f", text variable: GVL.trqOutputs[0]
    Textfield (562,101 72x30), "%.3f", text variable: GVL.motorDrive[0].kVirtual
        OnMouseClick: write the text variable via Default
    Textfield (384,375 72x30), "%.3f", text variable: GVL.motorDrive[6].trqOutput
    Textfield (384,417 72x30), "%.3f", text variable: GVL.motorDrive[7].trqOutput
    Textfield (384,456 72x30), "%.3f", text variable: GVL.motorDrive[8].trqOutput
    Textfield (385,555 72x30), "%.3f", text variable: GVL.motorDrive[10].trqOutput
    Textfield (385,595 72x30), "%.3f", text variable: GVL.motorDrive[11].trqOutput
    Textfield (472,141 72x30), "%.3f", text variable: GVL.trqOutputs[1]
    Textfield (472,182 72x30), "%.3f", text variable: GVL.trqOutputs[2]
    Textfield (473,242 72x30), "%.3f", text variable: GVL.trqOutputs[3]
    Textfield (473,281 72x30), "%.3f", text variable: GVL.trqOutputs[4]
    Textfield (473,321 72x30), "%.3f", text variable: GVL.trqOutputs[5]
    Textfield (474,515 72x30), "%.3f", text variable: GVL.trqOutputs[9]
    Textfield (473,375 72x30), "%.3f", text variable: GVL.trqOutputs[6]
    Textfield (473,417 72x30), "%.3f", text variable: GVL.trqOutputs[7]
    Textfield (473,456 72x30), "%.3f", text variable: GVL.trqOutputs[8]
    Textfield (474,555 72x30), "%.3f", text variable: GVL.trqOutputs[10]
    Textfield (474,595 72x30), "%.3f", text variable: GVL.trqOutputs[11]
    Textfield (562,141 72x30), "%.3f", text variable: GVL.motorDrive[1].kVirtual
        OnMouseClick: write the text variable via Default
    Textfield (562,182 72x30), "%.3f", text variable: GVL.motorDrive[2].kVirtual
        OnMouseClick: write the text variable via Default
    Textfield (563,242 72x30), "%.3f", text variable: GVL.motorDrive[3].kVirtual
        OnMouseClick: write the text variable via Default
    Textfield (563,281 72x30), "%.3f", text variable: GVL.motorDrive[4].kVirtual
        OnMouseClick: write the text variable via Default
    Textfield (563,321 72x30), "%.3f", text variable: GVL.motorDrive[5].kVirtual
        OnMouseClick: write the text variable via Default
    Textfield (564,515 72x30), "%.3f", text variable: GVL.motorDrive[9].kVirtual
        OnMouseClick: write the text variable via Default
    Textfield (563,375 72x30), "%.3f", text variable: GVL.motorDrive[6].kVirtual
        OnMouseClick: write the text variable via Default
    Textfield (563,417 72x30), "%.3f", text variable: GVL.motorDrive[7].kVirtual
        OnMouseClick: write the text variable via Default
    Textfield (563,456 72x30), "%.3f", text variable: GVL.motorDrive[8].kVirtual
        OnMouseClick: write the text variable via Default
    Textfield (564,555 72x30), "%.3f", text variable: GVL.motorDrive[10].kVirtual
        OnMouseClick: write the text variable via Default
    Textfield (564,595 72x30), "%.3f", text variable: GVL.motorDrive[11].kVirtual
        OnMouseClick: write the text variable via Default
    Textfield (651,141 72x30), "%.3f", text variable: GVL.motorDrive[1].bVirtual
        OnMouseClick: write the text variable via Default
    Textfield (651,182 72x30), "%.3f", text variable: GVL.motorDrive[2].bVirtual
        OnMouseClick: write the text variable via Default
    Textfield (652,242 72x30), "%.3f", text variable: GVL.motorDrive[3].bVirtual
        OnMouseClick: write the text variable via Default
    Textfield (652,281 72x30), "%.3f", text variable: GVL.motorDrive[4].bVirtual
        OnMouseClick: write the text variable via Default
    Textfield (652,321 72x30), "%.3f", text variable: GVL.motorDrive[5].bVirtual
        OnMouseClick: write the text variable via Default
    Textfield (653,515 72x30), "%.3f", text variable: GVL.motorDrive[9].bVirtual
        OnMouseClick: write the text variable via Default
    Textfield (652,375 72x30), "%.3f", text variable: GVL.motorDrive[6].bVirtual
        OnMouseClick: write the text variable via Default
    Textfield (652,417 72x30), "%.3f", text variable: GVL.motorDrive[7].bVirtual
        OnMouseClick: write the text variable via Default
    Textfield (652,456 72x30), "%.3f", text variable: GVL.motorDrive[8].bVirtual
        OnMouseClick: write the text variable via Default
    Textfield (653,555 72x30), "%.3f", text variable: GVL.motorDrive[10].bVirtual
        OnMouseClick: write the text variable via Default
    Textfield (653,595 72x30), "%.3f", text variable: GVL.motorDrive[11].bVirtual
        OnMouseClick: write the text variable via Default
    Textfield (739,141 72x30), "%.3f", text variable: GVL.motorDrive[1].kpTrqLoop
        OnMouseClick: write the text variable via Default
    Textfield (739,182 72x30), "%.3f", text variable: GVL.motorDrive[2].kpTrqLoop
        OnMouseClick: write the text variable via Default
    Textfield (740,242 72x30), "%.3f", text variable: GVL.motorDrive[3].kpTrqLoop
        OnMouseClick: write the text variable via Default
    Textfield (740,281 72x30), "%.3f", text variable: GVL.motorDrive[4].kpTrqLoop
        OnMouseClick: write the text variable via Default
    Textfield (740,321 72x30), "%.3f", text variable: GVL.motorDrive[5].kpTrqLoop
        OnMouseClick: write the text variable via Default
    Textfield (741,515 72x30), "%.3f", text variable: GVL.motorDrive[9].kpTrqLoop
        OnMouseClick: write the text variable via Default
    Textfield (740,375 72x30), "%.3f", text variable: GVL.motorDrive[6].kpTrqLoop
        OnMouseClick: write the text variable via Default
    Textfield (740,417 72x30), "%.3f", text variable: GVL.motorDrive[7].kpTrqLoop
        OnMouseClick: write the text variable via Default
    Textfield (740,456 72x30), "%.3f", text variable: GVL.motorDrive[8].kpTrqLoop
        OnMouseClick: write the text variable via Default
    Textfield (741,555 72x30), "%.3f", text variable: GVL.motorDrive[10].kpTrqLoop
        OnMouseClick: write the text variable via Default
    Textfield (741,595 72x30), "%.3f", text variable: GVL.motorDrive[11].kpTrqLoop
        OnMouseClick: write the text variable via Default
    Textfield (829,141 72x30), "%.3f", text variable: GVL.motorDrive[1].kiTrqLoop
        OnMouseClick: write the text variable via Default
    Textfield (829,182 72x30), "%.3f", text variable: GVL.motorDrive[2].kiTrqLoop
        OnMouseClick: write the text variable via Default
    Textfield (830,242 72x30), "%.3f", text variable: GVL.motorDrive[3].kiTrqLoop
        OnMouseClick: write the text variable via Default
    Textfield (830,281 72x30), "%.3f", text variable: GVL.motorDrive[4].kiTrqLoop
        OnMouseClick: write the text variable via Default
    Textfield (830,321 72x30), "%.3f", text variable: GVL.motorDrive[5].kiTrqLoop
        OnMouseClick: write the text variable via Default
    Textfield (831,515 72x30), "%.3f", text variable: GVL.motorDrive[9].kiTrqLoop
        OnMouseClick: write the text variable via Default
    Textfield (830,374 72x30), "%.3f", text variable: GVL.motorDrive[6].kiTrqLoop
        OnMouseClick: write the text variable via Default
    Textfield (830,417 72x30), "%.3f", text variable: GVL.motorDrive[7].kiTrqLoop
        OnMouseClick: write the text variable via Default
    Textfield (830,456 72x30), "%.3f", text variable: GVL.motorDrive[8].kiTrqLoop
        OnMouseClick: write the text variable via Default
    Textfield (831,555 72x30), "%.3f", text variable: GVL.motorDrive[10].kiTrqLoop
        OnMouseClick: write the text variable via Default
    Textfield (831,595 72x30), "%.3f", text variable: GVL.motorDrive[11].kiTrqLoop
        OnMouseClick: write the text variable via Default
    Textfield (918,141 72x30), "%.3f", text variable: GVL.motorDrive[1].reducerColbConstant
        OnMouseClick: write the text variable via Default
    Textfield (918,182 72x30), "%.3f", text variable: GVL.motorDrive[2].reducerColbConstant
        OnMouseClick: write the text variable via Default
    Textfield (919,242 72x30), "%.3f", text variable: GVL.motorDrive[3].reducerColbConstant
        OnMouseClick: write the text variable via Default
    Textfield (919,281 72x30), "%.3f", text variable: GVL.motorDrive[4].reducerColbConstant
        OnMouseClick: write the text variable via Default
    Textfield (919,321 72x30), "%.3f", text variable: GVL.motorDrive[5].reducerColbConstant
        OnMouseClick: write the text variable via Default
    Textfield (920,515 72x30), "%.3f", text variable: GVL.motorDrive[9].reducerColbConstant
        OnMouseClick: write the text variable via Default
    Textfield (919,375 72x30), "%.3f", text variable: GVL.motorDrive[6].reducerColbConstant
        OnMouseClick: write the text variable via Default
    Textfield (919,417 72x30), "%.3f", text variable: GVL.motorDrive[7].reducerColbConstant
        OnMouseClick: write the text variable via Default
    Textfield (919,456 72x30), "%.3f", text variable: GVL.motorDrive[8].reducerColbConstant
        OnMouseClick: write the text variable via Default
    Textfield (920,555 72x30), "%.3f", text variable: GVL.motorDrive[10].reducerColbConstant
        OnMouseClick: write the text variable via Default
    Textfield (920,595 72x30), "%.3f", text variable: GVL.motorDrive[11].reducerColbConstant
        OnMouseClick: write the text variable via Default
    Lamp1 (1101,143 27x29), variable: GVL.axisForceCtrlModeInd[1], style: Lamp-Lamp1-Green
    Lamp1 (1101,183 27x29), variable: GVL.axisForceCtrlModeInd[2], style: Lamp-Lamp1-Green
    Lamp1 (1101,244 27x29), variable: GVL.axisForceCtrlModeInd[3], style: Lamp-Lamp1-Green
    Lamp1 (1101,379 27x29), variable: GVL.axisForceCtrlModeInd[6], style: Lamp-Lamp1-Green
    Lamp1 (1101,283 27x29), variable: GVL.axisForceCtrlModeInd[4], style: Lamp-Lamp1-Green
    Lamp1 (1101,323 27x29), variable: GVL.axisForceCtrlModeInd[5], style: Lamp-Lamp1-Green
    Lamp1 (1101,418 27x29), variable: GVL.axisForceCtrlModeInd[7], style: Lamp-Lamp1-Green
    Lamp1 (1101,458 27x29), variable: GVL.axisForceCtrlModeInd[8], style: Lamp-Lamp1-Green
    Lamp1 (1101,518 27x29), variable: GVL.axisForceCtrlModeInd[9], style: Lamp-Lamp1-Green
    Lamp1 (1101,557 27x29), variable: GVL.axisForceCtrlModeInd[10], style: Lamp-Lamp1-Green
    Lamp1 (1101,597 27x29), variable: GVL.axisForceCtrlModeInd[11], style: Lamp-Lamp1-Green
    Lamp1 (81,106 27x29), variable: GVL.motorDrive[0].enableBit, style: Lamp-Lamp1-Green
    Lamp1 (81,145 27x29), variable: GVL.motorDrive[1].enableBit, style: Lamp-Lamp1-Green
    Lamp1 (81,185 27x29), variable: GVL.motorDrive[2].enableBit, style: Lamp-Lamp1-Green
    Lamp1 (81,245 27x29), variable: GVL.motorDrive[3].enableBit, style: Lamp-Lamp1-Green
    Lamp1 (81,378 27x29), variable: GVL.motorDrive[6].enableBit, style: Lamp-Lamp1-Green
    Lamp1 (81,284 27x29), variable: GVL.motorDrive[4].enableBit, style: Lamp-Lamp1-Green
    Lamp1 (81,324 27x29), variable: GVL.motorDrive[5].enableBit, style: Lamp-Lamp1-Green
    Lamp1 (81,417 27x29), variable: GVL.motorDrive[7].enableBit, style: Lamp-Lamp1-Green
    Lamp1 (81,457 27x29), variable: GVL.motorDrive[8].enableBit, style: Lamp-Lamp1-Green
    Lamp1 (81,516 27x29), variable: GVL.motorDrive[9].enableBit, style: Lamp-Lamp1-Green
    Lamp1 (81,555 27x29), variable: GVL.motorDrive[10].enableBit, style: Lamp-Lamp1-Green
    Lamp1 (81,595 27x29), variable: GVL.motorDrive[11].enableBit, style: Lamp-Lamp1-Green
    GroupBox (29,929 884x107), "Axis Group"
        Button (13,25 80x30), "Force Ctrl On"
            toggle GVL.forceCtrlGroupButton
        RadioButton (184,26 692x29), variable: GVL.groupSelector
            Areas[1]: Text=Shank
            Areas[2]: Text=Thigh
            Areas[3]: Text=Side
            Areas[4]: Text=LegA
            Areas[5]: Text=LegB
            Areas[6]: Text=LegC
            Areas[7]: Text=LegD
            Areas[8]: Text=LegE
            Areas[9]: Text=LegF
        Button (629,65 96x30), "Trq zero"
            toggle GVL.setTSRZeroButton
        Button (99,25 79x30), "Force Ctrl Off"
            toggle GVL.forceCtrlGroupOffButton
        Button (99,66 80x30), "Disable"
            toggle GVL.disableGroupButton
        Button (13,66 79x30), "Enable"
            toggle GVL.enableGroupButton
        Button (191,66 74x30), "Home"
            toggle GVL.homeGroupButton
        Button (276,66 74x30), "Set Pos"
            toggle GVL.setPosGroupButton
        Button (362,65 71x30), "Jog"
            toggle GVL.jogGroupButton
        Textfield (533,65 85x30), "%d", text variable: GVL.jogGroupVelocity
            OnMouseClick: write the text variable via Default
        Button (443,65 74x30), "Jog Stop"
            toggle GVL.jogStopGroupButton
    GroupBox (922,928 263x140), "Impedance Control"
        Textfield (13,19 72x30), "%.3f", text variable: GVL.kpGroup
            OnMouseClick: write the text variable via Default
        Textfield (97,19 72x30), "%.3f", text variable: GVL.kdGroup
            OnMouseClick: write the text variable via Default
        Textfield (98,59 72x30), "%.3f", text variable: GVL.kiTrqGroup
            OnMouseClick: write the text variable via Default
        Textfield (13,59 72x30), "%.3f", text variable: GVL.kpTrqGroup
            OnMouseClick: write the text variable via Default
        Button (183,19 73x30), "Hard"
            toggle GVL.useHardImpedButton
        Button (183,59 73x30), "Soft"
            toggle GVL.useSoftImpedButton
        Button (183,101 73x30), "Set Impd"
            toggle GVL.setGroupImpedButton
    Label (40,701 42x20), "E_T"
    Label (40,741 42x20), "E_A"
    Textfield (122,656 72x30), "%.3f", text variable: GVL.motorDrive[12].motorAngle
    Button (1010,656 74x30), "Force ctrl"
        toggle GVL.axisForceCtrlButton[12]
    Button (1010,696 74x30), "Force ctrl"
        toggle GVL.axisForceCtrlButton[13]
    Button (1010,736 74x30), "Force ctrl"
        toggle GVL.axisForceCtrlButton[14]
    Textfield (122,696 72x30), "%.3f", text variable: GVL.motorDrive[13].motorAngle
    Textfield (122,736 72x30), "%.3f", text variable: GVL.motorDrive[14].motorAngle
    Textfield (210,656 72x30), "%.2f", text variable: GVL.motorDrive[12].trqCalibrated
    Textfield (210,696 72x30), "%.2f", text variable: GVL.motorDrive[13].trqCalibrated
    Textfield (210,736 72x30), "%.2f", text variable: GVL.motorDrive[14].trqCalibrated
    Textfield (297,656 72x30), "%.3f", text variable: GVL.motorDrive[12].tgtAngle
        OnMouseClick: write the text variable via Default
    Textfield (297,696 72x30), "%.3f", text variable: GVL.motorDrive[13].tgtAngle
        OnMouseClick: write the text variable via Default
    Textfield (297,736 72x30), "%.3f", text variable: GVL.motorDrive[14].tgtAngle
        OnMouseClick: write the text variable via Default
    Textfield (385,656 72x30), "%.3f", text variable: GVL.motorDrive[12].trqOutput
    Textfield (385,696 72x30), "%.3f", text variable: GVL.motorDrive[13].trqOutput
    Textfield (385,736 72x30), "%.3f", text variable: GVL.motorDrive[14].trqOutput
    Textfield (474,656 72x30), "%.3f", text variable: GVL.trqOutputs[12]
    Textfield (474,696 72x30), "%.3f", text variable: GVL.trqOutputs[13]
    Textfield (474,736 72x30), "%.3f", text variable: GVL.trqOutputs[14]
    Textfield (564,656 72x30), "%.3f", text variable: GVL.motorDrive[12].kVirtual
        OnMouseClick: write the text variable via Default
    Textfield (564,696 72x30), "%.3f", text variable: GVL.motorDrive[13].kVirtual
        OnMouseClick: write the text variable via Default
    Textfield (564,736 72x30), "%.3f", text variable: GVL.motorDrive[14].kVirtual
        OnMouseClick: write the text variable via Default
    Textfield (653,656 72x30), "%.3f", text variable: GVL.motorDrive[12].bVirtual
        OnMouseClick: write the text variable via Default
    Textfield (653,696 72x30), "%.3f", text variable: GVL.motorDrive[13].bVirtual
        OnMouseClick: write the text variable via Default
    Textfield (653,736 72x30), "%.3f", text variable: GVL.motorDrive[14].bVirtual
        OnMouseClick: write the text variable via Default
    Textfield (741,656 72x30), "%.3f", text variable: GVL.motorDrive[12].kpTrqLoop
        OnMouseClick: write the text variable via Default
    Textfield (741,696 72x30), "%.3f", text variable: GVL.motorDrive[13].kpTrqLoop
        OnMouseClick: write the text variable via Default
    Textfield (741,736 72x30), "%.3f", text variable: GVL.motorDrive[14].kpTrqLoop
        OnMouseClick: write the text variable via Default
    Textfield (831,656 72x30), "%.3f", text variable: GVL.motorDrive[12].kiTrqLoop
        OnMouseClick: write the text variable via Default
    Textfield (831,696 72x30), "%.3f", text variable: GVL.motorDrive[13].kiTrqLoop
        OnMouseClick: write the text variable via Default
    Textfield (831,736 72x30), "%.3f", text variable: GVL.motorDrive[14].kiTrqLoop
        OnMouseClick: write the text variable via Default
    Textfield (920,656 72x30), "%.3f", text variable: GVL.motorDrive[12].reducerColbConstant
        OnMouseClick: write the text variable via Default
    Textfield (920,696 72x30), "%.3f", text variable: GVL.motorDrive[13].reducerColbConstant
        OnMouseClick: write the text variable via Default
    Textfield (920,736 72x30), "%.3f", text variable: GVL.motorDrive[14].reducerColbConstant
        OnMouseClick: write the text variable via Default
    Lamp1 (81,657 27x29), variable: GVL.motorDrive[12].enableBit, style: Lamp-Lamp1-Green
    Lamp1 (81,696 27x29), variable: GVL.motorDrive[13].enableBit, style: Lamp-Lamp1-Green
    Lamp1 (81,736 27x29), variable: GVL.motorDrive[14].enableBit, style: Lamp-Lamp1-Green
    Label (41,840 42x20), "F_T"
    Label (41,880 42x20), "F_A"
    Textfield (123,795 72x30), "%.3f", text variable: GVL.motorDrive[15].motorAngle
    Button (1011,795 74x30), "Force ctrl"
        toggle GVL.axisForceCtrlButton[15]
    Button (1011,835 74x30), "Force ctrl"
        toggle GVL.axisForceCtrlButton[16]
    Button (1011,875 74x30), "Force ctrl"
        toggle GVL.axisForceCtrlButton[17]
    Textfield (123,835 72x30), "%.3f", text variable: GVL.motorDrive[16].motorAngle
    Textfield (123,875 72x30), "%.3f", text variable: GVL.motorDrive[17].motorAngle
    Textfield (211,795 72x30), "%.2f", text variable: GVL.motorDrive[15].trqCalibrated
    Textfield (211,835 72x30), "%.2f", text variable: GVL.motorDrive[16].trqCalibrated
    Textfield (211,875 72x30), "%.2f", text variable: GVL.motorDrive[17].trqCalibrated
    Textfield (298,795 72x30), "%.3f", text variable: GVL.motorDrive[15].tgtAngle
        OnMouseClick: write the text variable via Default
    Textfield (298,835 72x30), "%.3f", text variable: GVL.motorDrive[16].tgtAngle
        OnMouseClick: write the text variable via Default
    Textfield (298,875 72x30), "%.3f", text variable: GVL.motorDrive[17].tgtAngle
        OnMouseClick: write the text variable via Default
    Textfield (386,795 72x30), "%.3f", text variable: GVL.motorDrive[15].trqOutput
    Textfield (386,835 72x30), "%.3f", text variable: GVL.motorDrive[16].trqOutput
    Textfield (386,875 72x30), "%.3f", text variable: GVL.motorDrive[17].trqOutput
    Textfield (475,795 72x30), "%.3f", text variable: GVL.trqOutputs[15]
    Textfield (475,835 72x30), "%.3f", text variable: GVL.trqOutputs[16]
    Textfield (475,875 72x30), "%.3f", text variable: GVL.trqOutputs[17]
    Textfield (565,795 72x30), "%.3f", text variable: GVL.motorDrive[15].kVirtual
        OnMouseClick: write the text variable via Default
    Textfield (565,835 72x30), "%.3f", text variable: GVL.motorDrive[16].kVirtual
        OnMouseClick: write the text variable via Default
    Textfield (565,875 72x30), "%.3f", text variable: GVL.motorDrive[17].kVirtual
        OnMouseClick: write the text variable via Default
    Textfield (654,795 72x30), "%.3f", text variable: GVL.motorDrive[15].bVirtual
        OnMouseClick: write the text variable via Default
    Textfield (654,835 72x30), "%.3f", text variable: GVL.motorDrive[16].bVirtual
        OnMouseClick: write the text variable via Default
    Textfield (654,875 72x30), "%.3f", text variable: GVL.motorDrive[17].bVirtual
        OnMouseClick: write the text variable via Default
    Textfield (742,795 72x30), "%.3f", text variable: GVL.motorDrive[15].kpTrqLoop
        OnMouseClick: write the text variable via Default
    Textfield (742,835 72x30), "%.3f", text variable: GVL.motorDrive[16].kpTrqLoop
        OnMouseClick: write the text variable via Default
    Textfield (742,875 72x30), "%.3f", text variable: GVL.motorDrive[17].kpTrqLoop
        OnMouseClick: write the text variable via Default
    Textfield (832,795 72x30), "%.3f", text variable: GVL.motorDrive[15].kiTrqLoop
        OnMouseClick: write the text variable via Default
    Textfield (832,835 72x30), "%.3f", text variable: GVL.motorDrive[16].kiTrqLoop
        OnMouseClick: write the text variable via Default
    Textfield (832,875 72x30), "%.3f", text variable: GVL.motorDrive[17].kiTrqLoop
        OnMouseClick: write the text variable via Default
    Textfield (921,795 72x30), "%.3f", text variable: GVL.motorDrive[15].reducerColbConstant
        OnMouseClick: write the text variable via Default
    Textfield (921,835 72x30), "%.3f", text variable: GVL.motorDrive[16].reducerColbConstant
        OnMouseClick: write the text variable via Default
    Textfield (921,875 72x30), "%.3f", text variable: GVL.motorDrive[17].reducerColbConstant
        OnMouseClick: write the text variable via Default
    Lamp1 (82,796 27x29), variable: GVL.motorDrive[15].enableBit, style: Lamp-Lamp1-Green
    Lamp1 (82,835 27x29), variable: GVL.motorDrive[16].enableBit, style: Lamp-Lamp1-Green
    Lamp1 (82,875 27x29), variable: GVL.motorDrive[17].enableBit, style: Lamp-Lamp1-Green
    Lamp1 (1101,699 27x29), variable: GVL.axisForceCtrlModeInd[13], style: Lamp-Lamp1-Green
    Lamp1 (1101,739 27x29), variable: GVL.axisForceCtrlModeInd[14], style: Lamp-Lamp1-Green
END_VISUALIZATION

// ---- VISUs/Monitor.TcVIS
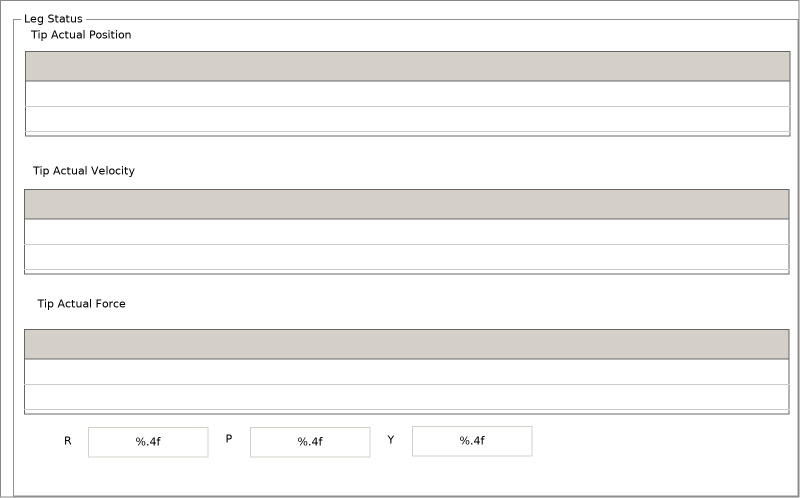
VISUALIZATION Monitor  // 800x498
    GroupBox (13,11 785x485), "Leg Status"
        Table (12,40 765x85), data array: GVL.tipActualPos
            p3854506369: GVL.tipActualPos[0,INDEX]
            p1892666644: GVL.tipActualPos[1,INDEX]
            p338671338: GVL.tipActualPos[2,INDEX]
            p2170511999: GVL.tipActualPos[3,INDEX]
            p3723444502: GVL.tipActualPos[4,INDEX]
            p1218418051: GVL.tipActualPos[5,INDEX]
            p2232123230: LegA
            p511219082: LegB
            p1755163831: LegC
            p4092479075: LegD
            p2237128397: LegE
            p505689113: LegF
        Table (11,178 765x85), data array: GVL.tipActualVel
            p3854506369: GVL.tipActualVel[0,INDEX]
            p1892666644: GVL.tipActualVel[1,INDEX]
            p338671338: GVL.tipActualVel[2,INDEX]
            p2170511999: GVL.tipActualVel[3,INDEX]
            p3723444502: GVL.tipActualVel[4,INDEX]
            p1218418051: GVL.tipActualVel[5,INDEX]
            p2232123230: LegA
            p511219082: LegB
            p1755163831: LegC
            p4092479075: LegD
            p2237128397: LegE
            p505689113: LegF
        Label (16,9 105x30), "Tip Actual Position"
        Label (6,145 130x30), "Tip Actual Velocity"
        Label (20,278 115x30), "Tip Actual Force"
        Table (11,318 765x85), data array: GVL.tipActualFce
            p3854506369: GVL.tipActualFce[0,INDEX]
            p1892666644: GVL.tipActualFce[1,INDEX]
            p338671338: GVL.tipActualFce[2,INDEX]
            p2170511999: GVL.tipActualFce[3,INDEX]
            p3723444502: GVL.tipActualFce[4,INDEX]
            p1218418051: GVL.tipActualFce[5,INDEX]
            p2232123230: LegA
            p511219082: LegB
            p1755163831: LegC
            p4092479075: LegD
            p2237128397: LegE
            p505689113: LegF
        Textfield (75,416 120x30), "%.4f", text variable: GVL.rpy_model[0]
        Textfield (237,416 120x30), "%.4f", text variable: GVL.rpy_model[1]
        Textfield (399,415 120x30), "%.4f", text variable: GVL.rpy_model[2]
        Label (356,414 44x30), "Y"
        Label (194,413 44x30), "P"
        Label (33,415 44x30), "R"
END_VISUALIZATION

